(* Start Stop Motor *)

PROGRAM main
  VAR
    Start_PB : BOOL;
    Stop_PB : BOOL;
    Motor : BOOL;
  END_VAR

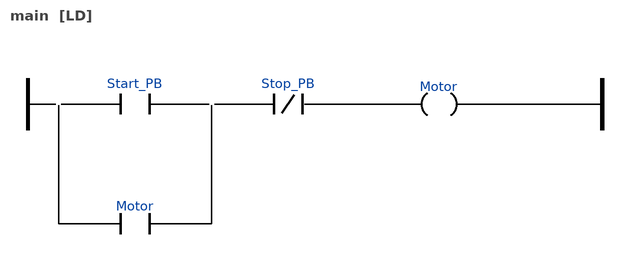
(* LD diagram, written out as Structured Text *)
Motor := (Motor OR Start_PB) AND NOT Stop_PB;
END_PROGRAM
